// Mitsubishi GX Works2 project: 888888   PLC: FX3U/FX3UC

PROGRAM MAIN
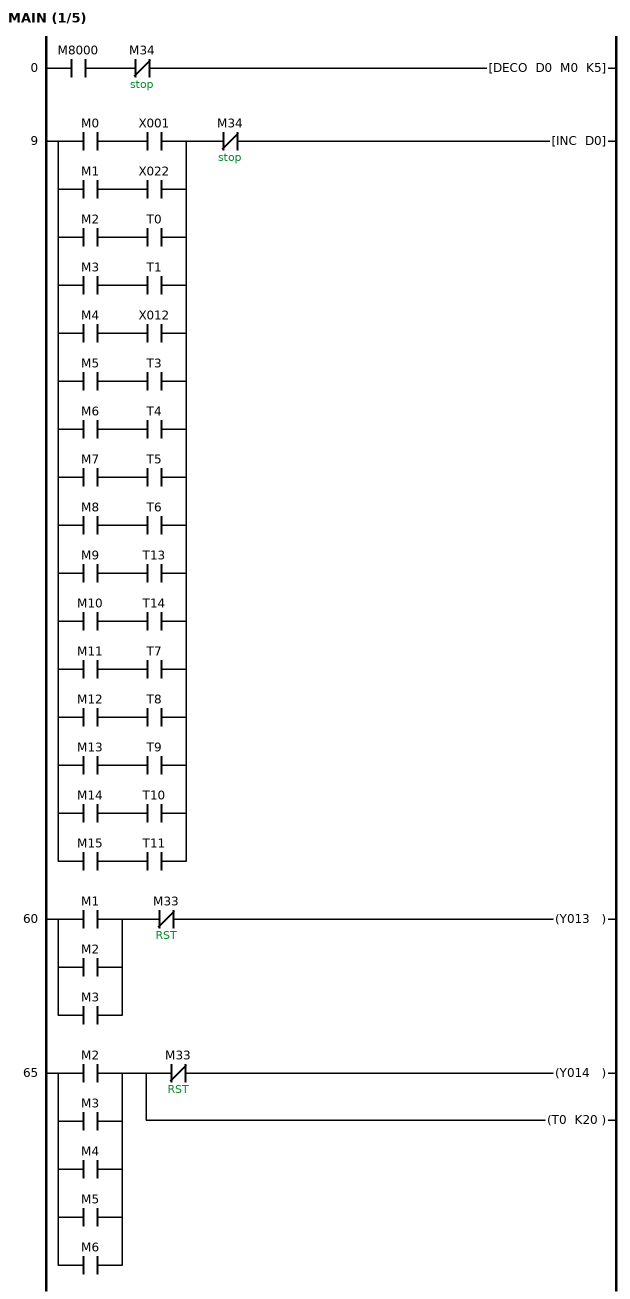
0     LD      M8000
      ANI     M34  ; stop
      DECO    D0 M0 K5
9     LD      M0
      AND     X001
      LD      M1
      AND     X022
      ORB
      LD      M2
      AND     T0
      ORB
      LD      M3
      AND     T1
      ORB
      LD      M4
      AND     X012
      ORB
      LD      M5
      AND     T3
      ORB
      LD      M6
      AND     T4
      ORB
      LD      M7
      AND     T5
      ORB
      LD      M8
      AND     T6
      ORB
      LD      M9
      AND     T13
      ORB
      LD      M10
      AND     T14
      ORB
      LD      M11
      AND     T7
      ORB
      LD      M12
      AND     T8
      ORB
      LD      M13
      AND     T9
      ORB
      LD      M14
      AND     T10
      ORB
      LD      M15
      AND     T11
      ORB
      ANI     M34  ; stop
      INC     D0
60    LD      M1
      OR      M2
      OR      M3
      ANI     M33  ; RST
      OUT     Y013
65    LD      M2
      OR      M3
      OR      M4
      OR      M5
      OR      M6
      MPS
      ANI     M33  ; RST
      OUT     Y014
      MPP
      OUT     T0 K20
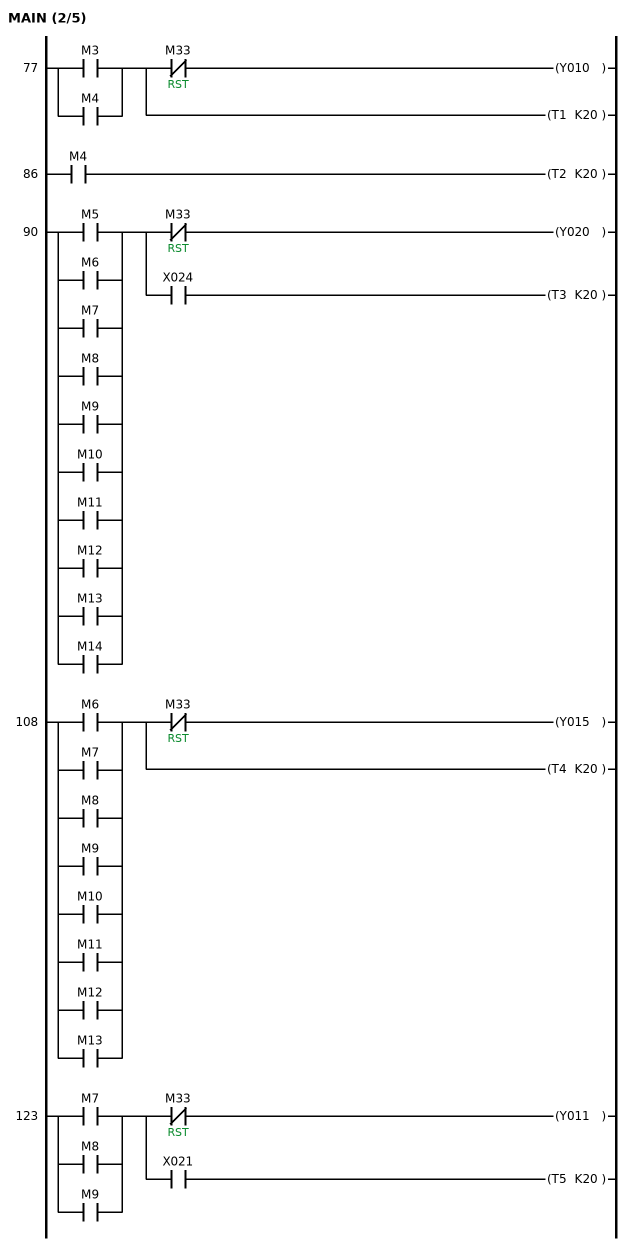
77    LD      M3
      OR      M4
      MPS
      ANI     M33  ; RST
      OUT     Y010
      MPP
      OUT     T1 K20
86    LD      M4
      OUT     T2 K20
90    LD      M5
      OR      M6
      OR      M7
      OR      M8
      OR      M9
      OR      M10
      OR      M11
      OR      M12
      OR      M13
      OR      M14
      MPS
      ANI     M33  ; RST
      OUT     Y020
      MPP
      AND     X024
      OUT     T3 K20
108   LD      M6
      OR      M7
      OR      M8
      OR      M9
      OR      M10
      OR      M11
      OR      M12
      OR      M13
      MPS
      ANI     M33  ; RST
      OUT     Y015
      MPP
      OUT     T4 K20
123   LD      M7
      OR      M8
      OR      M9
      MPS
      ANI     M33  ; RST
      OUT     Y011
      MPP
      AND     X021
      OUT     T5 K20
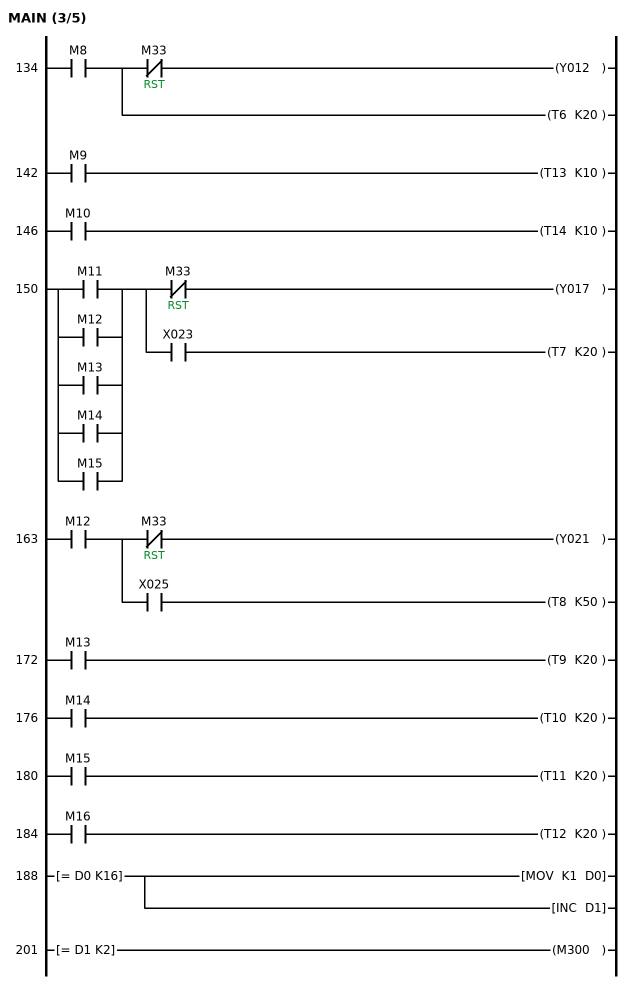
134   LD      M8
      MPS
      ANI     M33  ; RST
      OUT     Y012
      MPP
      OUT     T6 K20
142   LD      M9
      OUT     T13 K10
146   LD      M10
      OUT     T14 K10
150   LD      M11
      OR      M12
      OR      M13
      OR      M14
      OR      M15
      MPS
      ANI     M33  ; RST
      OUT     Y017
      MPP
      AND     X023
      OUT     T7 K20
163   LD      M12
      MPS
      ANI     M33  ; RST
      OUT     Y021
      MPP
      AND     X025
      OUT     T8 K50
172   LD      M13
      OUT     T9 K20
176   LD      M14
      OUT     T10 K20
180   LD      M15
      OUT     T11 K20
184   LD      M16
      OUT     T12 K20
188   LD=     D0 K16
      MOV     K1 D0
      INC     D1
201   LD=     D1 K2
      OUT     M300
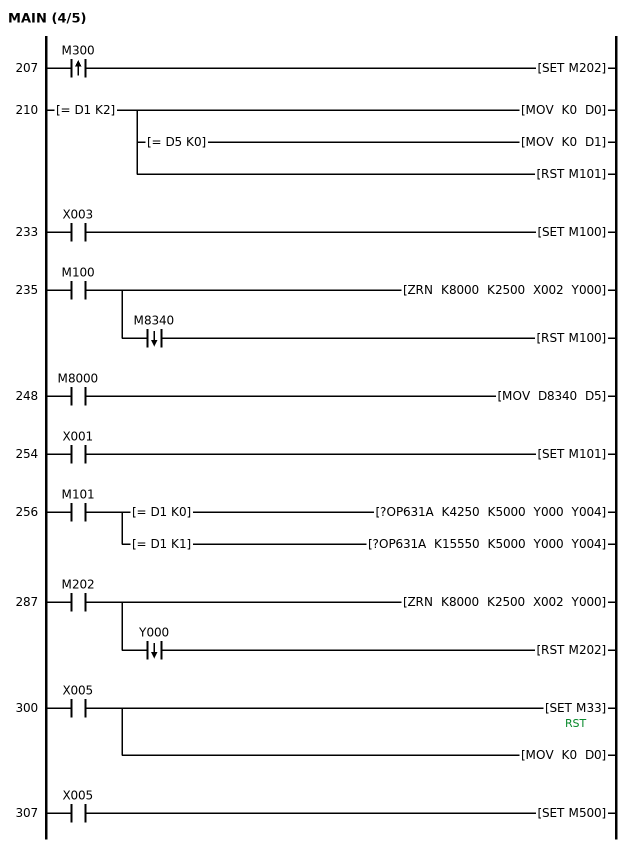
207   LDP     M300
      SET     M202
210   LD=     D1 K2
      MOV     K0 D0
      MPS
      AND=    D5 K0
      MOV     K0 D1
      MPP
      RST     M101
233   LD      X003
      SET     M100
235   LD      M100
      ZRN     K8000 K2500 X002 Y000
      ANDF    M8340
      RST     M100
248   LD      M8000
      MOV     D8340 D5
254   LD      X001
      SET     M101
256   LD      M101
      MPS
      AND=    D1 K0
      ?OP631A K4250 K5000 Y000 Y004
      MPP
      AND=    D1 K1
      ?OP631A K15550 K5000 Y000 Y004
287   LD      M202
      ZRN     K8000 K2500 X002 Y000
      ANDF    Y000
      RST     M202
300   LD      X005
      SET     M33  ; RST
      MOV     K0 D0
307   LD      X005
      SET     M500
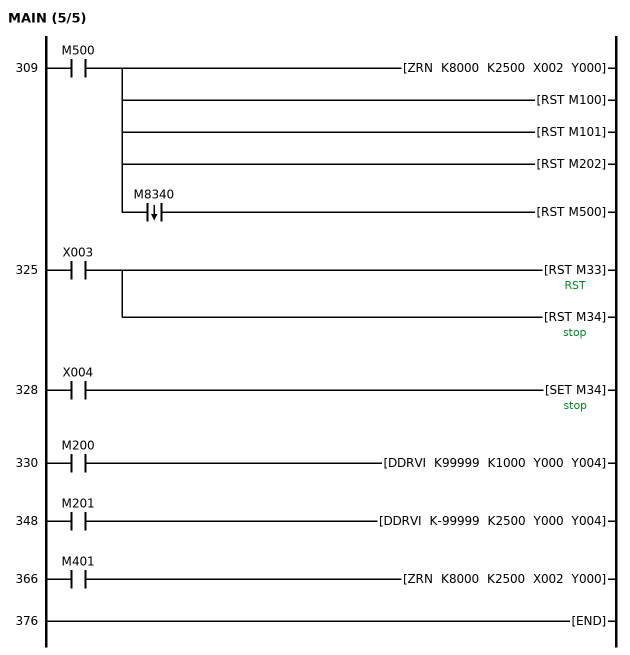
309   LD      M500
      ZRN     K8000 K2500 X002 Y000
      RST     M100
      RST     M101
      RST     M202
      ANDF    M8340
      RST     M500
325   LD      X003
      RST     M33  ; RST
      RST     M34  ; stop
328   LD      X004
      SET     M34  ; stop
330   LD      M200
      DDRVI   K99999 K1000 Y000 Y004
348   LD      M201
      DDRVI   K-99999 K2500 Y000 Y004
366   LD      M401
      ZRN     K8000 K2500 X002 Y000
376   END
END_PROGRAM
